// TIA Portal V18 export
VAR_GLOBAL   // PLC tag table "Cabinet_10"
   Sz10_Button_LED_ST11_ST12 AT %Q2000.0 : Bool;
   Sz10_Button_LED_ST12_ST13 AT %Q2000.1 : Bool;
   "Reserved(146)" AT %Q2000.2 : Bool;
   "Reserved(147)" AT %Q2000.3 : Bool;
   "Reserved(148)" AT %Q2000.4 : Bool;
   "Reserved(149)" AT %Q2000.5 : Bool;
   "Reserved(150)" AT %Q2000.6 : Bool;
   "Reserved(151)" AT %Q2000.7 : Bool;
   Sz10_ST11_SenA AT %I2000.0 : Bool;
   Sz10_ST11_SenB AT %I2000.1 : Bool;
   Sz10_ST11_SenC AT %I2000.2 : Bool;
   Sz10_ST11_SenD AT %I2000.3 : Bool;
   Sz10_ST12_SenA AT %I2000.4 : Bool;
   Sz10_ST12_SenB AT %I2000.5 : Bool;
   Sz10_ST12_SenC AT %I2000.6 : Bool;
   Sz10_ST12_SenD AT %I2000.7 : Bool;
   Sz10_Button_ST11_ST12 AT %I2001.0 : Bool;
   Sz10_Button_ST12_ST13 AT %I2001.1 : Bool;
   "Reserved(152)" AT %I2001.2 : Bool;
   "Reserved(153)" AT %I2001.3 : Bool;
   "Reserved(154)" AT %I2001.4 : Bool;
   "Reserved(155)" AT %I2001.5 : Bool;
   "Reserved(156)" AT %I2001.6 : Bool;
   "Reserved(157)" AT %I2001.7 : Bool;
   Sz10_Safety1_1 AT %I2050.0 : Bool;
   "Reserved(158)" AT %I2050.1 : Bool;
   "Reserved(159)" AT %I2050.2 : Bool;
   "Reserved(160)" AT %I2050.3 : Bool;
   Sz10_Safety1_2 AT %I2050.4 : Bool;
   "Reserved(161)" AT %I2050.5 : Bool;
   "Reserved(162)" AT %I2050.6 : Bool;
   "Reserved(163)" AT %I2050.7 : Bool;
   "Reserved(171)" AT %I2051.0 : Bool;
   "Reserved(170)" AT %I2051.1 : Bool;
   "Reserved(169)" AT %I2051.2 : Bool;
   "Reserved(168)" AT %I2051.3 : Bool;
   "Reserved(167)" AT %I2051.4 : Bool;
   "Reserved(166)" AT %I2051.5 : Bool;
   "Reserved(165)" AT %I2051.6 : Bool;
   "Reserved(164)" AT %I2051.7 : Bool;
END_VAR
